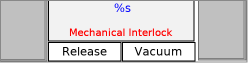
VISUALIZATION Std_VacuumVal_Ctrl  // 248x63
VAR_IN_OUT
	m_Input_Inst : None;
END_VAR
    RoundedRectangle (48,0 146x41), "%s", text variable: m_Input_Inst.IN_Name
    RoundedRectangle (48,42 73x19), "Release", colour toggle: (m_Input_Inst.S_Release) <> 0, invisible if: (m_Input_Inst.E_PurgeErr) <> 0
    RoundedRectangle (122,42 73x19), "Vacuum", colour toggle: (m_Input_Inst.S_Vacuum) <> 0, invisible if: (m_Input_Inst.E_VacuumErr) <> 0
    Group (-1,0 46x59)
        tap m_Input_Inst.T_ManPurge
        Button (0,0 48x61)
            tap m_Input_Inst.In_ManHome
        Polygon (38,51)
        Polygon (35,51)
    Group (198,0 46x59)
        tap m_Input_Inst.T_ManVacuum
        Button (0,0 48x60)
            tap m_Input_Inst.In_ManWork
        Polygon (10,50)
        Polygon (13,50)
    RoundedRectangle (48,23 146x19), "Mechanical Interlock", invisible if: (NOT (NOT m_Input_Inst.In_VacuumX AND m_Input_Inst.T_ManVacuum)) <> 0
    RoundedRectangle (48,23 146x19), "Mechanical Interlock", invisible if: (NOT (NOT m_Input_Inst.In_PurgeX AND m_Input_Inst.T_ManPurge)) <> 0
    RoundedRectangle (48,42 73x19), "Release", colour toggle: (m_Input_Inst.E_PurgeErr) <> 0, invisible if: (NOT m_Input_Inst.E_PurgeErr) <> 0
    RoundedRectangle (122,42 73x19), "Vacuum", colour toggle: (m_Input_Inst.E_VacuumErr) <> 0, invisible if: (NOT m_Input_Inst.E_VacuumErr) <> 0
END_VISUALIZATION

(* stored: Version 1.1.0.1, ProductVersion 3.1.4018.2
   Visu Std_VacuumVal_Ctrl: Id {f6d3ba12-21cb-4842-95b2-230aae12ad4e} *)
